(* IEC 61131-3 sources: beckhoffAutomationInterface/ST/Shark/Lib/ErrorHandling, 14 files *)

(* ---- E_ErrorId.st ---- *)
(* Unified error code enumeration for the library. *)
{attribute 'qualified_only'}
{attribute 'strict'}
{attribute 'to_string'}
TYPE E_ErrorId :
    (
        NO_ERROR := 0,

        // General / System (1000+)
        ERR_GEN_INTERNAL                := 1000,
        ERR_GEN_INVALID_PARAM           := 1001,
        ERR_GEN_NULL_POINTER            := 1002,
        ERR_GEN_TIMEOUT                 := 1003,
        ERR_GEN_NOT_IMPLEMENTED         := 1004,
        ERR_GEN_INITIALIZATION          := 1005,
        ERR_GEN_NOT_CONFIGURED          := 1006, // POU executed before Configure() was called

        ERR_HW_SENSOR_OPEN              := 2000, // Wire break / Open circuit
        ERR_HW_SENSOR_SHORT             := 2001, // Short circuit
        ERR_HW_SENSOR_OVERRANGE         := 2002, // Value > Max physical limit
        ERR_HW_SENSOR_UNDERRANGE        := 2003, // Value < Min physical limit
        ERR_HW_OUTPUT_FAULT             := 2010, // Digital/Analog output failure
        ERR_HW_POWER_SUPPLY             := 2020,
        ERR_HW_MOTION_FAULT             := 2030, // Axis motion fault (homing/move/stop) — phase in context

        ERR_CTRL_LIMIT_EXCEEDED         := 3000, // Process Value > Safety Limit
        ERR_CTRL_DEVIATION_HIGH         := 3001, // PV deviates from SP > Tolerance
        ERR_CTRL_WATCHDOG_HEATING       := 3002, // Heating active but Temp dropping
        ERR_CTRL_WATCHDOG_COOLING       := 3003, // Cooling active but Temp rising
        ERR_CTRL_TUNING_ERROR           := 3004,
        ERR_CTRL_FAULT                  := 3005, // Controller reported a generic fault
        ERR_CTRL_SAFETY_TRIPPED         := 3006, // TwinSAFE / system-level safety not OK

        ERR_COMM_PORT_CLOSED            := 4000, // Serial port not open
        ERR_COMM_TIMEOUT                := 4001, // No response from slave
        ERR_COMM_CRC_ERROR              := 4002, // Checksum mismatch
        ERR_COMM_BUFFER_OVERFLOW        := 4003, // Receive buffer full
        ERR_COMM_FRAME_ERROR            := 4004, // Invalid frame format
        ERR_COMM_PROTOCOL               := 4005, // Protocol-level error
        ERR_COMM_INVALID_RESPONSE       := 4006, // Invalid or unexpected response
        ERR_COMM_DATA_CONVERSION        := 4007, // Data conversion failed
        ERR_COMM_MODBUS_EXCEPTION       := 4010, // Slave returned Modbus Exception
        ERR_COMM_ETHERCAT_STATE         := 4020,

        ERR_DEV_BRONKHORST_FAULT        := 5000, // Bronkhorst specific error bit
        ERR_DEV_HARDWARE_ERROR          := 5030, // Generic device hardware error
        ERR_DEVICE_NACK                 := 5040, // Device returned NACK

        ERR_VALVE_NOT_CONFIGURED        := 6000, // Valve not configured
        ERR_VALVE_INVALID_INDEX         := 6001, // Invalid output index
        ERR_VALVE_FEEDBACK_TIMEOUT      := 6002, // Feedback not received in time
        ERR_VALVE_FEEDBACK_MISMATCH     := 6003, // Feedback doesn't match command

        // Behavior Tree Errors (7000+)
        ERR_BT_NULL_INTERFACE           := 7000, // Interface not configured
        ERR_BT_NULL_CHILD               := 7001, // Child node not set
        ERR_BT_CHILD_FAILED             := 7002, // Child node returned failure
        ERR_BT_SEQUENCE_FAILED          := 7003, // Sequence node failed
        ERR_BT_SENSOR_ERROR             := 7004, // Sensor reported error
        ERR_BT_VALVE_ERROR              := 7005, // Valve reported error
        ERR_BT_CONDITION_FAILED         := 7006, // Condition check failed
        ERR_BT_TIMEOUT                  := 7007, // Operation timed out
        ERR_BT_MAX_RETRIES              := 7008, // Maximum retry attempts exceeded
        ERR_BT_MAX_CHILDREN             := 7009, // Maximum children exceeded
        ERR_BT_PARALLEL_FAILED          := 7010, // Parallel node failure threshold reached
        ERR_BT_FORCED_FAILURE           := 7011, // FB_AlwaysFailureNode / ForceFailure decorator
        ERR_BT_CONDITION_NOT_CONFIGURED := 7012  // FB_ConditionNode reference not set
    ) UDINT;
END_TYPE

(* ---- E_EventId.st ---- *)
(* Non-error event identifiers for the library (operational / informational logs). *)
{attribute 'qualified_only'}
{attribute 'strict'}
{attribute 'to_string'}
TYPE E_EventId :
    (
        NONE := 0,

        // Generic informational / diagnostic event; free text carried in the log
        // context. Use when a message does not need its own filterable ID.
        // Specific IDs (command lifecycle, state changes, etc.) are added per
        // call site during migration, in non-overlapping bands above 10000
        // (E_ErrorId occupies 0..7999).
        EVT_INFO := 10000
    ) UDINT;
END_TYPE

(* ---- E_TcEventSeverity.st ---- *)
{attribute 'qualified_only'}
{attribute 'strict'}
TYPE E_TcEventSeverity :
    (
        Verbose  := 0,
        Info     := 1,
        Warning  := 2,
        Error    := 3,
        Critical := 4
    )INT;
END_TYPE

(* ---- ST_Error.st ---- *)
(* Standard error information structure. *)
TYPE ST_Error :
STRUCT
    eErrorId         : E_ErrorId          := E_ErrorId.NO_ERROR;
    eSeverity        : E_TcEventSeverity  := E_TcEventSeverity.Error;
    sSource          : STRING(80);        // Component that currently owns the error
    sMessage         : STRING(255);       // Description (may include chained child sources)
    fCurrentValue    : REAL;              // Optional measured value (RaiseWithValues), exported in JSON
    fExpectedValue   : REAL;              // Optional limit/setpoint (RaiseWithValues), exported in JSON
    sUnits           : STRING(15);        // Optional units for the values (e.g. 'C', 'bar')
    tTimestamp       : DT;                // Time most recent propagation/raise occurred
    tOriginTimestamp : DT;                // Time the root cause first occurred (preserved across RaiseFromChild)
END_STRUCT
END_TYPE

(* ---- GVL_ErrorLogger.st ---- *)
{attribute 'qualified_only'}
VAR_GLOBAL
    Logger : FB_ErrorLogger; // Global singleton for error logging
END_VAR

(* ---- GVL_EventLogger.st ---- *)
(* TC3 EventLogger integration: console-trace switch. *)
{attribute 'qualified_only'}
VAR_GLOBAL
    // Master switch for the parallel ADSLOG console trace in FB_TcEventLoggerSink.
    // The TC3 EventLogger is always the primary sink. Keep TRUE while verifying
    // the EventLogger path in XAE; set FALSE to make the EventLogger the sole sink.
    bConsoleTrace : BOOL := TRUE;
END_VAR

(* ---- I_Errorable.st ---- *)
(* Base interface for components that can report errors. *)
INTERFACE I_Errorable EXTENDS __System.IQueryInterface

METHOD IsError : BOOL
END_METHOD

METHOD GetError : ST_Error
END_METHOD

END_INTERFACE

(* ---- I_LogSink.st ---- *)
(* Transport abstraction for the logging facade (FB_ErrorLogger).
   A sink receives a fully-resolved log record and is responsible ONLY for
   getting it out (TC3 EventLogger, ADSLOG console trace, a test spy, a
   machine-specific transport, ...).
   Swapping the sink lets a machine or a test change the transport without
   touching the logging policy/throttle in FB_ErrorLogger / FB_ErrorHandler. *)
INTERFACE I_LogSink

METHOD Publish
VAR_INPUT
    sSource       : STRING(255);            // Emitting source (POU/method) for HMI source info
    nEventId      : UDINT;                  // E_ErrorId / E_EventId value
    sId           : STRING(80);             // Human-readable id (for the console trace)
    sContext      : STRING(255);            // Dynamic detail (sensor reading, command, ...)
    eSeverity     : E_TcEventSeverity;
    fCurrentValue : REAL := 0;              // Optional measured value, exported in the JSON attribute
    fExpectedValue: REAL := 0;              // Optional limit/setpoint, exported in the JSON attribute
    sUnits        : STRING(15) := '';       // Optional units for the values
END_VAR
END_METHOD

END_INTERFACE

(* ---- F_FormatIso8601.st ---- *)
(* Formats a Date-Time (DT) value as an ISO-8601 string 'YYYY-MM-DDThh:mm:ss'.
   Used for the tTimestamp field of the EventLogger JSON attribute so clients
   get the same timestamp shape the legacy logger emitted.

   Implementation: TwinCAT DT_TO_STRING yields the fixed-width IEC form
   'DT#YYYY-MM-DD-hh:mm:ss'. We strip the 'DT#' prefix and replace the single
   '-' separator between the date and the time (position 11) with a 'T'.
   The DT resolution is one second, matching the legacy timestamp. *)
FUNCTION F_FormatIso8601 : STRING(19)
VAR_INPUT
    dtIn : DT;
END_VAR
VAR
    sTmp  : STRING(40);
    nHash : INT;
END_VAR
    sTmp := DT_TO_STRING(dtIn);          // 'DT#YYYY-MM-DD-hh:mm:ss'
    nHash := FIND(sTmp, '#');
    IF nHash > 0 THEN
        sTmp := DELETE(sTmp, nHash, 1);  // remove the 'DT#' prefix -> 'YYYY-MM-DD-hh:mm:ss'
    END_IF
    sTmp := REPLACE(sTmp, 'T', 1, 11);   // date/time separator '-' -> 'T'
    F_FormatIso8601 := sTmp;
END_FUNCTION

(* ---- F_FormatLimitError.st ---- *)
(* Formats a limit error message with value and limit. *)
FUNCTION F_FormatLimitError : STRING(255)
VAR_INPUT
    sLabel  : STRING(20);   // Error label (e.g., 'Temp', 'Deviation')
    rActual : LREAL;        // Actual value
    rLimit  : LREAL;        // Limit value
    sUnit   : STRING(10);   // Unit (e.g., 'C', '%')
END_VAR
VAR
    sResult : STRING(255);
END_VAR
    sResult := CONCAT(sLabel, ' ');
    sResult := CONCAT(sResult, LREAL_TO_FMTSTR(rActual, 2, TRUE));
    sResult := CONCAT(sResult, sUnit);
    sResult := CONCAT(sResult, ' > limit ');
    sResult := CONCAT(sResult, LREAL_TO_FMTSTR(rLimit, 2, TRUE));
    sResult := CONCAT(sResult, sUnit);

    F_FormatLimitError := sResult;
END_FUNCTION

(* ---- F_GetCurrentDT.st ---- *)
(* Returns the current system time as a Date-Time (DT) value. *)
FUNCTION F_GetCurrentDT : DT
VAR
    fbGetTime  : GETSYSTEMTIME;
    stFileTime : T_FILETIME;
END_VAR
    // Get current system time (100ns ticks since 1601)
    fbGetTime(timeLoDW => stFileTime.dwLowDateTime, timeHiDW => stFileTime.dwHighDateTime);

    // Convert to Date-Time (Seconds since 1970)
    F_GetCurrentDT := FILETIME_TO_DT(stFileTime);
END_FUNCTION

(* ---- FB_ErrorHandler.st ---- *)
(* Centralized error handling component for raising and managing errors. *)
FUNCTION_BLOCK FB_ErrorHandler
VAR
    _stError : ST_Error;
    _sSourceName : STRING(80);
    // Heartbeat throttle: re-log a persistent fault at most once per interval
    // (T#0S disables the heartbeat: first occurrence + clear only).
    _tHeartbeatInterval : TIME := T#1M;
    _tLastLogTime : DT;
    _nOccurrenceCount : UDINT;
END_VAR

METHOD PUBLIC Init : BOOL
VAR_INPUT
    sSourceName        : STRING(80);
    tHeartbeatInterval : TIME := T#1M;
END_VAR
    _sSourceName := sSourceName;
    _tHeartbeatInterval := tHeartbeatInterval;
    Clear();
    Init := TRUE;
END_METHOD

METHOD PUBLIC Raise
VAR_INPUT
    eErrorId  : E_ErrorId;
    sMessage  : STRING(255);
    eSeverity : E_TcEventSeverity := E_TcEventSeverity.Error;
END_VAR
    IF eErrorId = E_ErrorId.NO_ERROR THEN
        RETURN;
    END_IF

    // Same fault still active: count it and heartbeat periodically,
    // instead of flooding every cycle or going silent forever.
    IF _stError.eErrorId = eErrorId THEN
        _HandleRepeat();
        RETURN;
    END_IF

    _ApplyError(eErrorId := eErrorId, sMessage := sMessage, eSeverity := eSeverity);
END_METHOD

METHOD PUBLIC RaiseWithValues
VAR_INPUT
    eErrorId  : E_ErrorId;
    sLabel    : STRING(20);
    rActual   : LREAL;
    rLimit    : LREAL;
    sUnit     : STRING(10);
    eSeverity : E_TcEventSeverity := E_TcEventSeverity.Error;
END_VAR
VAR
    sMessage : STRING(255);
END_VAR
    IF eErrorId = E_ErrorId.NO_ERROR THEN
        RETURN;
    END_IF

    // Same fault still active: count it and heartbeat periodically,
    // instead of flooding every cycle or going silent forever.
    IF _stError.eErrorId = eErrorId THEN
        _HandleRepeat();
        RETURN;
    END_IF

    sMessage := F_FormatLimitError(sLabel, rActual, rLimit, sUnit);
    _ApplyError(eErrorId := eErrorId, sMessage := sMessage, eSeverity := eSeverity,
                fCurrentValue := TO_REAL(rActual), fExpectedValue := TO_REAL(rLimit), sUnits := sUnit);
END_METHOD

    (* Raises an error from a child component, chaining the source for traceability.
       Preserves the child's origin timestamp and severity. *)
METHOD PUBLIC RaiseFromChild
VAR_INPUT
    stChildError : ST_Error;
END_VAR
VAR
    sChainedMsg : STRING(255);
END_VAR
    IF stChildError.eErrorId = E_ErrorId.NO_ERROR THEN
        RETURN;
    END_IF

    // Prevent cyclic spamming of string manipulation
    IF _stError.eErrorId = stChildError.eErrorId THEN
        RETURN;
    END_IF

    sChainedMsg := LEFT(CONCAT(CONCAT('[', stChildError.sSource), CONCAT('] ', stChildError.sMessage)), 255);

    _stError.eErrorId := stChildError.eErrorId;
    _stError.eSeverity := stChildError.eSeverity;
    _stError.sSource := _sSourceName;
    _stError.sMessage := sChainedMsg;
    _stError.fCurrentValue := stChildError.fCurrentValue;
    _stError.fExpectedValue := stChildError.fExpectedValue;
    _stError.sUnits := stChildError.sUnits;
    _stError.tTimestamp := F_GetCurrentDT();
    // Preserve the root-cause occurrence time from the child when available,
    // so forensics at subsystem level can still see when the fault first hit.
    IF stChildError.tOriginTimestamp <> DT#1970-01-01-00:00:00 THEN
        _stError.tOriginTimestamp := stChildError.tOriginTimestamp;
    ELSE
        _stError.tOriginTimestamp := _stError.tTimestamp;
    END_IF
    _nOccurrenceCount := 1;
    _tLastLogTime := _stError.tTimestamp;
    // Do NOT re-log here: the error was already logged when it originated.
    // Propagation only carries state up the tree.
END_METHOD

METHOD PRIVATE _ApplyError
VAR_INPUT
    eErrorId      : E_ErrorId;
    sMessage      : STRING(255);
    eSeverity     : E_TcEventSeverity;
    fCurrentValue : REAL := 0;
    fExpectedValue: REAL := 0;
    sUnits        : STRING(15) := '';
END_VAR
VAR
    tNow : DT;
END_VAR
    tNow := F_GetCurrentDT();
    _stError.eErrorId := eErrorId;
    _stError.eSeverity := eSeverity;
    _stError.sSource := _sSourceName;
    _stError.sMessage := sMessage;
    _stError.fCurrentValue := fCurrentValue;
    _stError.fExpectedValue := fExpectedValue;
    _stError.sUnits := sUnits;
    _stError.tTimestamp := tNow;
    _stError.tOriginTimestamp := tNow;
    _nOccurrenceCount := 1;
    _tLastLogTime := tNow;
    _LogError(sMessage);
END_METHOD

METHOD PRIVATE _LogError
VAR_INPUT
    sContext : STRING(255);
END_VAR
    GVL_ErrorLogger.Logger.LogError(
        sSource := _sSourceName,
        eErrorId := _stError.eErrorId,
        sContext := sContext,
        eSeverity := _stError.eSeverity,
        fCurrentValue := _stError.fCurrentValue,
        fExpectedValue := _stError.fExpectedValue,
        sUnits := _stError.sUnits
    );
END_METHOD

    (* Handles a re-raise of the currently active fault: counts the occurrence and
       re-logs at most once per heartbeat interval so a persistent fault stays
       visible without flooding the log every scan cycle. *)
METHOD PRIVATE _HandleRepeat
VAR
    tNow         : DT;
    nElapsedSec  : DWORD;
    nIntervalSec : DWORD;
END_VAR
    _nOccurrenceCount := _nOccurrenceCount + 1;

    nIntervalSec := TIME_TO_DWORD(_tHeartbeatInterval) / 1000;
    IF nIntervalSec = 0 THEN
        RETURN; // Heartbeat disabled: first occurrence + clear only.
    END_IF

    tNow := F_GetCurrentDT();
    nElapsedSec := DT_TO_DWORD(tNow) - DT_TO_DWORD(_tLastLogTime);
    IF nElapsedSec >= nIntervalSec THEN
        _stError.tTimestamp := tNow;
        _LogHeartbeat();
        _tLastLogTime := tNow;
    END_IF
END_METHOD

    (* Re-logs the active fault with its occurrence count (heartbeat). *)
METHOD PRIVATE _LogHeartbeat
VAR
    sContext : STRING(255);
END_VAR
    sContext := CONCAT('still active (', UDINT_TO_STRING(_nOccurrenceCount));
    sContext := CONCAT(sContext, 'x): ');
    sContext := LEFT(CONCAT(sContext, _stError.sMessage), 255);
    GVL_ErrorLogger.Logger.LogError(
        sSource := _sSourceName,
        eErrorId := _stError.eErrorId,
        sContext := sContext,
        eSeverity := _stError.eSeverity,
        fCurrentValue := _stError.fCurrentValue,
        fExpectedValue := _stError.fExpectedValue,
        sUnits := _stError.sUnits
    );
END_METHOD

    (* Logs a one-line resolution summary when an active fault clears. *)
METHOD PRIVATE _LogCleared
VAR
    sContext : STRING(255);
END_VAR
    sContext := CONCAT('cleared after ', UDINT_TO_STRING(_nOccurrenceCount));
    sContext := CONCAT(sContext, ' occurrence(s)');
    GVL_ErrorLogger.Logger.LogError(
        sSource := _sSourceName,
        eErrorId := _stError.eErrorId,
        sContext := sContext,
        eSeverity := E_TcEventSeverity.Info,
        fCurrentValue := _stError.fCurrentValue,
        fExpectedValue := _stError.fExpectedValue,
        sUnits := _stError.sUnits
    );
END_METHOD

METHOD PUBLIC Clear
    // Emit a one-line resolution summary when an active fault clears, so the
    // log records when and after how many occurrences it recovered.
    IF _stError.eErrorId <> E_ErrorId.NO_ERROR THEN
        _LogCleared();
    END_IF

    _stError.eErrorId := E_ErrorId.NO_ERROR;
    _stError.eSeverity := E_TcEventSeverity.Error;
    _stError.sSource := '';
    _stError.sMessage := '';
    _stError.fCurrentValue := 0;
    _stError.fExpectedValue := 0;
    _stError.sUnits := '';
    _stError.tTimestamp := DT#1970-01-01-00:00:00;
    _stError.tOriginTimestamp := DT#1970-01-01-00:00:00;
    _nOccurrenceCount := 0;
    _tLastLogTime := DT#1970-01-01-00:00:00;
END_METHOD

METHOD PUBLIC IsActive : BOOL
    IsActive := _stError.eErrorId <> E_ErrorId.NO_ERROR;
END_METHOD

METHOD PUBLIC GetError : ST_Error
    GetError := _stError;
END_METHOD

METHOD PUBLIC GetErrorId : E_ErrorId
    GetErrorId := _stError.eErrorId;
END_METHOD

END_FUNCTION_BLOCK

(* ---- FB_ErrorLogger.st ---- *)
(* Global logger. Single funnel for all library logging (errors + events).
   Owns logging POLICY only (the LogError/LogEvent/LogInfo API + id/severity
   resolution); the actual transport is delegated to an I_LogSink. The sink
   defaults to the built-in FB_TcEventLoggerSink and can be replaced via
   SetSink (e.g. a test spy or a machine-specific transport).
   Deduplication/throttling is handled by callers (e.g. FB_ErrorHandler). *)
FUNCTION_BLOCK FB_ErrorLogger
VAR
    _fbDefaultSink : FB_TcEventLoggerSink; // Built-in transport (TC3 EventLogger + console trace)
    _ipSink        : I_LogSink;            // Active transport; defaults to _fbDefaultSink
END_VAR

METHOD PUBLIC LogError : BOOL
VAR_INPUT
    sSource       : STRING(255);
    eErrorId      : E_ErrorId;
    sContext      : STRING(255);
    eSeverity     : E_TcEventSeverity := E_TcEventSeverity.Error;
    fCurrentValue : REAL := 0;          // Optional: measured value, exported in the event JSON attribute
    fExpectedValue: REAL := 0;          // Optional: limit/setpoint, exported in the event JSON attribute
    sUnits        : STRING(15) := '';   // Optional: units for the values (e.g. 'sccm', 'bar')
END_VAR

    IF eErrorId = E_ErrorId.NO_ERROR THEN
        RETURN;
    END_IF

    _Emit(sSource := sSource, nEventId := TO_UDINT(eErrorId), sId := TO_STRING(eErrorId), sContext := sContext, eSeverity := eSeverity,
          fCurrentValue := fCurrentValue, fExpectedValue := fExpectedValue, sUnits := sUnits);
    LogError := TRUE;
END_METHOD

    (* Logs a non-error operational event (severity defaults to Info). *)
METHOD PUBLIC LogEvent : BOOL
VAR_INPUT
    sSource    : STRING(255);
    eEventId   : E_EventId;
    sContext   : STRING(255);
    eSeverity  : E_TcEventSeverity := E_TcEventSeverity.Info;
END_VAR

    _Emit(sSource := sSource, nEventId := TO_UDINT(eEventId), sId := TO_STRING(eEventId), sContext := sContext, eSeverity := eSeverity);
    LogEvent := TRUE;
END_METHOD

    (* Logs a generic informational message (free text, no specific event ID). *)
METHOD PUBLIC LogInfo : BOOL
VAR_INPUT
    sSource  : STRING(255);
    sContext : STRING(255);
END_VAR

    _Emit(sSource := sSource, nEventId := TO_UDINT(E_EventId.EVT_INFO), sId := TO_STRING(E_EventId.EVT_INFO), sContext := sContext, eSeverity := E_TcEventSeverity.Info);
    LogInfo := TRUE;
END_METHOD

    (* Shared sink: resolves the active transport (defaulting to the built-in
       TC3 EventLogger sink) and publishes the record. This is the single point
       that controls all logging. *)
METHOD PRIVATE _Emit
VAR_INPUT
    sSource       : STRING(255);
    nEventId      : UDINT;
    sId           : STRING(80);
    sContext      : STRING(255);
    eSeverity     : E_TcEventSeverity;
    fCurrentValue : REAL := 0;
    fExpectedValue: REAL := 0;
    sUnits        : STRING(15) := '';
END_VAR
    // Lazily bind the default sink so the logger is never null and works out of
    // the box; SetSink can override it before or after first use.
    IF _ipSink = 0 THEN
        _ipSink := _fbDefaultSink;
    END_IF

    _ipSink.Publish(sSource := sSource, nEventId := nEventId, sId := sId,
                    sContext := sContext, eSeverity := eSeverity,
                    fCurrentValue := fCurrentValue, fExpectedValue := fExpectedValue, sUnits := sUnits);
END_METHOD

    (* Overrides the transport sink (e.g. a test spy or a machine-specific
       transport). A null sink is ignored so logging is never broken. *)
METHOD PUBLIC SetSink
VAR_INPUT
    ipSink : I_LogSink;
END_VAR
    IF ipSink <> 0 THEN
        _ipSink := ipSink;
    END_IF
END_METHOD

END_FUNCTION_BLOCK

(* ---- FB_TcEventLoggerSink.st ---- *)
(* Default log sink: TwinCAT 3 EventLogger transport, plus an optional ADSLOG
   console trace gated by GVL_EventLogger.bConsoleTrace.

   This is the built-in sink used by FB_ErrorLogger out of the box. Swap it via
   FB_ErrorLogger.SetSink to redirect logging (e.g. a test spy or a
   machine-specific transport) without changing any logging policy.

   NOTE: requires the Tc3_EventLogger and Tc3_JsonXml library references and an
   event class named BeckhoffLibEvents registered in XAE, holding one event per
   severity (Verbose, Info, Warning, Error, Critical). Each event text uses two
   indexed insertions, '{0} - {1}', for the error id and the dynamic context.
   TwinCAT substitutes arguments by zero-based index ({0}, {1}) — NOT printf '%s'.
   Each event also carries a JSON attribute so HMI/clients can read structured
   values directly. The attribute keeps the legacy logger's field names for
   client back-compat — {sComponentName, eErrorId, sErrorMessage, fCurrentValue,
   fExpectedValue, sUnits, tTimestamp} — and appends two new fields:
   sErrorIdText (the symbolic error-id name) and eSeverity (numeric severity). *)
FUNCTION_BLOCK FB_TcEventLoggerSink IMPLEMENTS I_LogSink
VAR
    _fbMessage    : FB_TcMessage;        // TC3 EventLogger message
    _fbSourceInfo : FB_TcSourceInfo;     // Carries the emitting source so the HMI can distinguish same-id events
    _fbJson       : FB_JsonSaxWriter;    // Builds the per-event JSON attribute consumed by HMI/clients
END_VAR

METHOD Publish
VAR_INPUT
    sSource       : STRING(255);
    nEventId      : UDINT;
    sId           : STRING(80);
    sContext      : STRING(255);
    eSeverity     : E_TcEventSeverity;
    fCurrentValue : REAL := 0;
    fExpectedValue: REAL := 0;
    sUnits        : STRING(15) := '';
END_VAR
VAR
    sFullMsg   : STRING(255);
    nMsgType   : DWORD;
    stEntry    : TcEventEntry;
    sJson      : STRING(800);
    sTimestamp : STRING(19);
    hr         : HRESULT;
END_VAR
    // 1) Optional console trace (ADSLOG), gated by a global switch. The TC3
    //    EventLogger (below) is the primary sink; this is for live tracing.
    IF GVL_EventLogger.bConsoleTrace THEN
        CASE eSeverity OF
            E_TcEventSeverity.Verbose,
            E_TcEventSeverity.Info:
                nMsgType := ADSLOG_MSGTYPE_HINT;
            E_TcEventSeverity.Warning:
                nMsgType := ADSLOG_MSGTYPE_WARN;
            E_TcEventSeverity.Error,
            E_TcEventSeverity.Critical:
                nMsgType := ADSLOG_MSGTYPE_ERROR;
        ELSE
            nMsgType := ADSLOG_MSGTYPE_ERROR;
        END_CASE
        sFullMsg := CONCAT(CONCAT(sSource, ': '), CONCAT(sId, ' - '));
        sFullMsg := CONCAT(sFullMsg, sContext);
        ADSLOGSTR(nMsgType, '%s', sFullMsg);
    END_IF

    // 2) TC3 EventLogger (persistent; consumed by the HMI over ADS). Severity
    //    selects one of five registered events in the BeckhoffLibEvents class;
    //    the event text and severity come from that registration. sSource is
    //    attached as source info so the HMI shows which POU/hardware raised it,
    //    and sId + sContext are passed as message arguments so the registered
    //    text can carry the dynamic detail via indexed insertions ('{0} - {1}').
    CASE eSeverity OF
        E_TcEventSeverity.Verbose:
            stEntry := TC_EVENTS.BeckhoffLibEvents.Verbose;
        E_TcEventSeverity.Info:
            stEntry := TC_EVENTS.BeckhoffLibEvents.Info;
        E_TcEventSeverity.Warning:
            stEntry := TC_EVENTS.BeckhoffLibEvents.Warning;
        E_TcEventSeverity.Error:
            stEntry := TC_EVENTS.BeckhoffLibEvents.Error;
        E_TcEventSeverity.Critical:
            stEntry := TC_EVENTS.BeckhoffLibEvents.Critical;
    ELSE
        stEntry := TC_EVENTS.BeckhoffLibEvents.Error;
    END_CASE

    // Clear() resets stale fields before reuse — this single source-info instance
    // is shared across every source, so without it a prior source's data could leak.
    _fbSourceInfo.Clear();
    _fbSourceInfo.sName := sSource;
    hr := _fbMessage.CreateEx(stEntry, _fbSourceInfo);
    IF _fbMessage.ipArguments <> 0 THEN
        _fbMessage.ipArguments.Clear();
        _fbMessage.ipArguments.AddString(sId);
        _fbMessage.ipArguments.AddString(sContext);
    END_IF
    // Attach the full record as the event JSON attribute so HMI/clients get every
    // detail in one place. The first seven keys keep the legacy logger's names
    // and order for client back-compat; sErrorIdText and eSeverity are appended
    // as new, additive fields so existing parsers keep working.
    sTimestamp := F_FormatIso8601(F_GetCurrentDT());   // AddString takes its arg by reference, so it needs a writable variable
    _fbJson.ResetDocument();
    _fbJson.StartObject();
    _fbJson.AddKey('sComponentName');  _fbJson.AddString(sSource);
    _fbJson.AddKey('eErrorId');        _fbJson.AddUdint(nEventId);
    _fbJson.AddKey('sErrorMessage');   _fbJson.AddString(sContext);
    _fbJson.AddKey('fCurrentValue');   _fbJson.AddReal(fCurrentValue);
    _fbJson.AddKey('fExpectedValue');  _fbJson.AddReal(fExpectedValue);
    _fbJson.AddKey('sUnits');          _fbJson.AddString(sUnits);
    _fbJson.AddKey('tTimestamp');      _fbJson.AddString(sTimestamp);
    _fbJson.AddKey('sErrorIdText');    _fbJson.AddString(sId);
    _fbJson.AddKey('eSeverity');       _fbJson.AddDint(TO_DINT(eSeverity));
    _fbJson.EndObject();
    _fbJson.CopyDocument(sJson, SIZEOF(sJson));
    _fbMessage.SetJsonAttribute(sJson);
    hr := _fbMessage.Send(0);
END_METHOD

END_FUNCTION_BLOCK
